Universal Robots PolyScope program: xmlrpc_example.urp

Program xmlrpc_example (installation=default directory=/home/ur/ursim-current/programs createdIn=3.1.16828.0 lastSavedIn=5.3.0.6470 robotSerialNumber=20183599999)
Calibrated DH parameters: a=[0, -0.425, -0.3922, 0, 0, 0]; d=[0.1625, 0, 0, 0.1333, 0.0997, 0.0996]; alpha=[1.570796, 0, 0, 1.570796, -1.570796, 0]; deltaTheta=[0, 0, 0, 0, 0, 0]
BeforeStart
  camera := rpc_factory("xmlrpc","http://127.0.0.1:50000")
Robot Program (runOnlyOnce=false)
  next_pose := camera.get_next_pose(Joint_6_name)
  MoveJ speed 60 deg/s, acceleration 80 deg/s^2 (useActiveTCP=true) feature=Base
    Waypoint Waypoint (Variable): variable=next_pose
  Halt
